// TIA Portal V20 export
TYPE "MABS_Setpoint"
// stored: Access Published, Namespace LineD1
   STRUCT
      ChangeBallsDirection : Bool;   // 0=forward; 1=backward
      Speed_balls : Int := 0;   // Based on preset speed setting. 60/70/80/90 m/min.
      Init_offset : Int;   // Offset angle for initial position -8/+10°
   END_STRUCT;
END_TYPE
